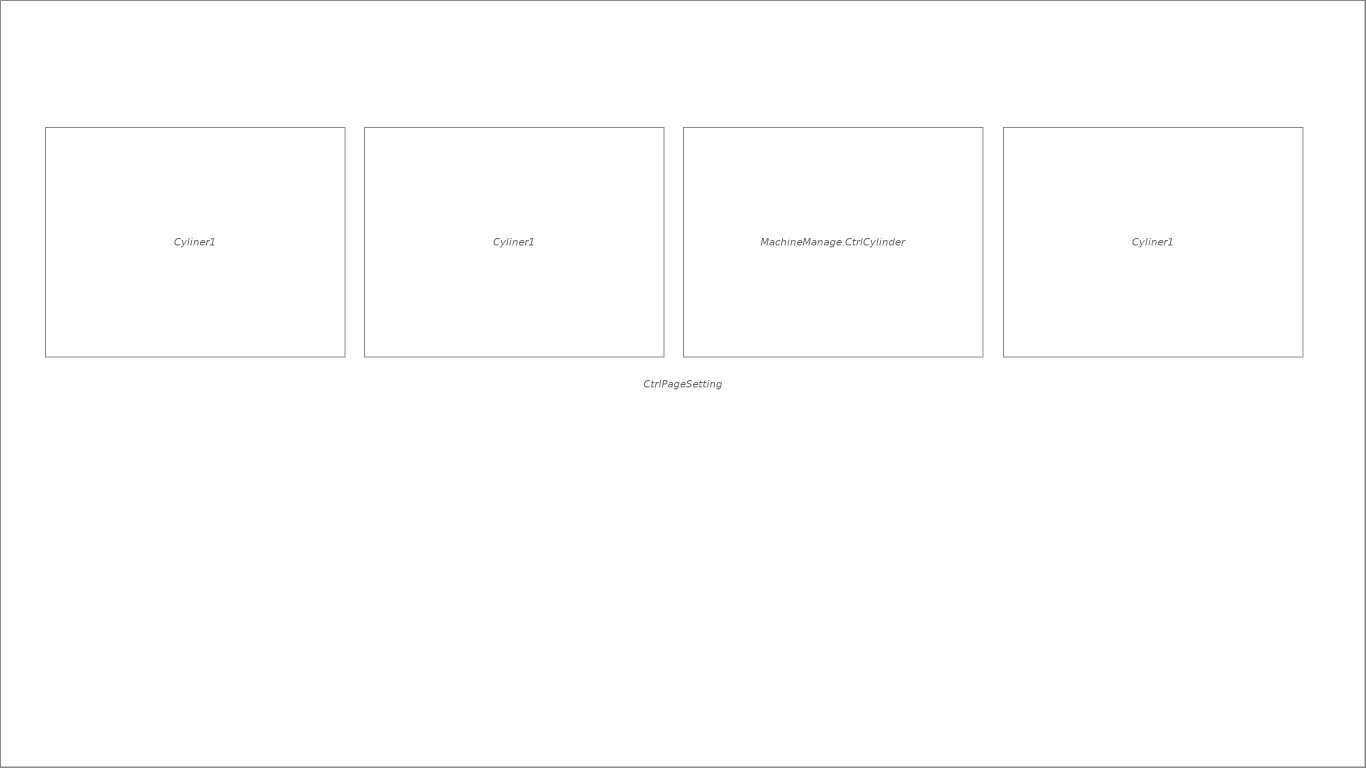
VISUALIZATION PageSetting_Steering  // 1366x768
    Frame (0,0 1366x768)
        shows CtrlPageSetting()
    Frame (45,127 300x230)
        shows Cyliner1(System := G_stSystem, Cylinder := G_arrCylinder[E_Cylinder.SteeringLift], CylinderData := G_arrCylinderData[E_Cylinder.SteeringLift])
    Frame (364,127 300x230)
        shows Cyliner1(System := G_stSystem, Cylinder := G_arrCylinder[E_Cylinder.SteeringAcquireElevator], CylinderData := G_arrCylinderData[E_Cylinder.SteeringAcquireElevator])
    Frame (683,127 300x230)
        shows MachineManage.CtrlCylinder(System := G_stSystem, Cylinder := G_arrCylinder[E_Cylinder.SteeringRotate], CylinderData := G_arrCylinderData[E_Cylinder.SteeringRotate])
    Frame (1003,127 300x230)
        shows Cyliner1(System := G_stSystem, Cylinder := G_arrCylinder[E_Cylinder.SteeringAcquireLimit], CylinderData := G_arrCylinderData[E_Cylinder.SteeringAcquireLimit])
END_VISUALIZATION

(* stored: Version 1.1.0.1, ProductVersion 3.1.4024.3
   Visu PageSetting_Steering: Id {38e739f2-8f0e-40d2-acfa-2962238b88f0} *)
